(* CODESYS project CODESYS_BLOG_AmazonAlexa_Example.project

Project tree, tasks and I/O mapping:
  Device : CODESYS Control Win V3 x64, 3S - Smart Software Solutions GmbH, version 3.5.12.0
    application Application
      libraries: Standard, * (System)
      task MainTask (cyclic, interval t#20ms, priority 1) calls PLC_PRG
      program PLC_PRG [ST]
      global variables GVL
      Symbols
*)

// Device/Application/GVL

VAR_GLOBAL
	bStartJob:BOOL:=FALSE;
	uiProductionCode:INT:=0;
	uiNumberOfScrews:INT:=0;
END_VAR

// Device/Application/PLC_PRG
PROGRAM PLC_PRG
VAR
END_VAR

bStartJob;
uiProductionCode;
uiNumberOfScrews;

END_PROGRAM
